(* CODESYS project elevator_project.project

Project tree, tasks and I/O mapping:
  Device : CODESYS Control Win V3, 3S - Smart Software Solutions GmbH, order no. 305021, version 3.5.9.40
    application Application
      libraries: Standard, * (System)
      task MainTask (cyclic, interval t#20ms, priority 1) calls PLC_PRG
      task VISU_TASK (cyclic, interval 100 ms, priority 31) calls VisuElems.Visu_Prg
      program PLC_PRG [SFC]: Init_entry, Init_active, GoTo_active, Idle_entry, Idle_exit, UpdateDesireFloor_active, UP_entry, DOWN_entry, UP_active, DOWN_active, Idle_active, Listener
      global variables GVL
      visualisation Visualization
  libraries: VisuSymbols, 3.5.8.0 (System)
  text list GlobalTextList
*)

// Device/Application/GVL
{attribute 'qualified_only'}
VAR_GLOBAL
	AtLevel1: BOOL;
	AtLevel2: BOOL;
	AtLevel3: BOOL;
	
	overweight: BOOL;
	
	Bottom: BOOL;
	Top: BOOL;
	
	Call1: BOOL;
	Call2: BOOL;
	Call3: BOOL;
	
	GoLevel1: BOOL;
	GoLevel2: BOOL;
	GoLevel3: BOOL;
	
	goDown: BOOL;
	goUp: BOOL;
	
	// Code
	calls: ARRAY[1..3] OF BOOL;
	i: INT;
	
	NOKButton: BOOL;
	goingUp: BOOL;
	goingDown: BOOL;
	desiredFloor: INT:=1;
	currentFloor: INT:=2;
	MAXFLOOR: INT:=3;
	
	useless: BOOL;
	
	openDahDoor: BOOL;
	arrived: BOOL;
	
	Done: BOOL;
	
	// State
	InitOk: BOOL;
	busy: BOOL;
	emergency: BOOL;
	request: BOOL;
END_VAR

// Device/Application/PLC_PRG
PROGRAM PLC_PRG
VAR
END_VAR
VAR // added by the converter: edge detectors and wires of the graphical bodies
    _w1, _w3, _w5, _w6, _w8, _w9, _w10, _w11 : BOOL;
    _w2, _w4, _w7 : INT;
END_VAR

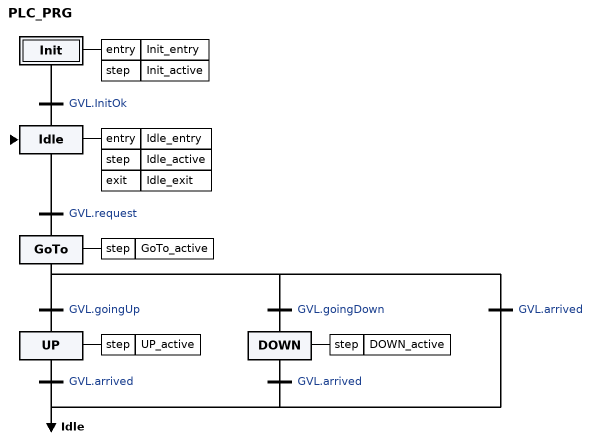
INITIAL_STEP Init:
    Init_entry(P1);  // entry action
    Init_active(N);  // step action
END_STEP
TRANSITION FROM Init TO Idle
    := GVL.InitOk;
END_TRANSITION
STEP Idle:
    Idle_entry(P1);  // entry action
    Idle_active(N);  // step action
    Idle_exit(P0);  // exit action
END_STEP
TRANSITION FROM Idle TO GoTo
    := GVL.request;
END_TRANSITION
STEP GoTo:
    GoTo_active(N);  // step action
END_STEP
TRANSITION FROM GoTo TO UP
    := GVL.goingUp;
END_TRANSITION
STEP UP:
    UP_active(N);  // step action
END_STEP
TRANSITION FROM UP TO Idle
    := GVL.arrived;
END_TRANSITION
TRANSITION FROM GoTo TO DOWN
    := GVL.goingDown;
END_TRANSITION
STEP DOWN:
    DOWN_active(N);  // step action
END_STEP
TRANSITION FROM DOWN TO Idle
    := GVL.arrived;
END_TRANSITION
TRANSITION FROM GoTo TO Idle
    := GVL.arrived;
END_TRANSITION

ACTION Init_entry:
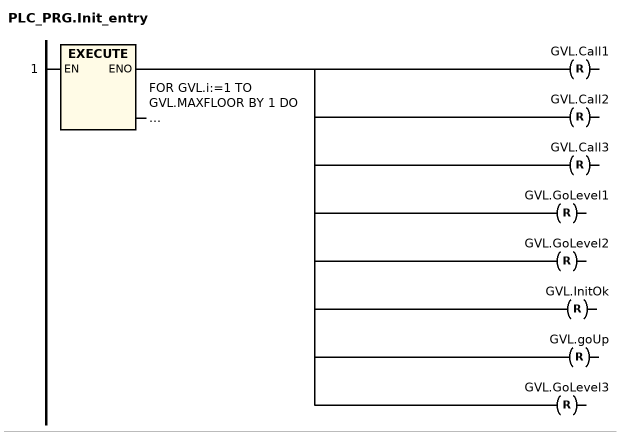
// NETWORK 1
FOR GVL.i:=1 TO GVL.MAXFLOOR BY 1 DO
	GVL.calls[GVL.i]:=FALSE;
END_FOR;
GVL.Call1 R= TRUE;
GVL.Call2 R= TRUE;
GVL.Call3 R= TRUE;
GVL.GoLevel1 R= TRUE;
GVL.GoLevel2 R= TRUE;
GVL.InitOk R= TRUE;
GVL.goUp R= TRUE;
GVL.GoLevel3 R= TRUE;
END_ACTION

ACTION Init_active:
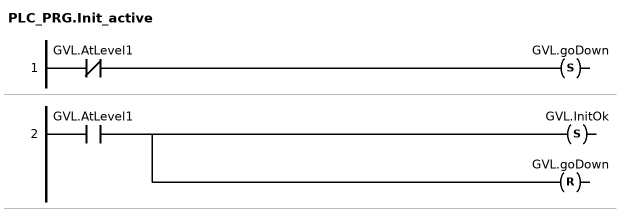
// NETWORK 1
GVL.goDown S= NOT GVL.AtLevel1;

// NETWORK 2
_w1 := GVL.AtLevel1;
GVL.InitOk S= _w1;
GVL.goDown R= _w1;
END_ACTION

ACTION GoTo_active:
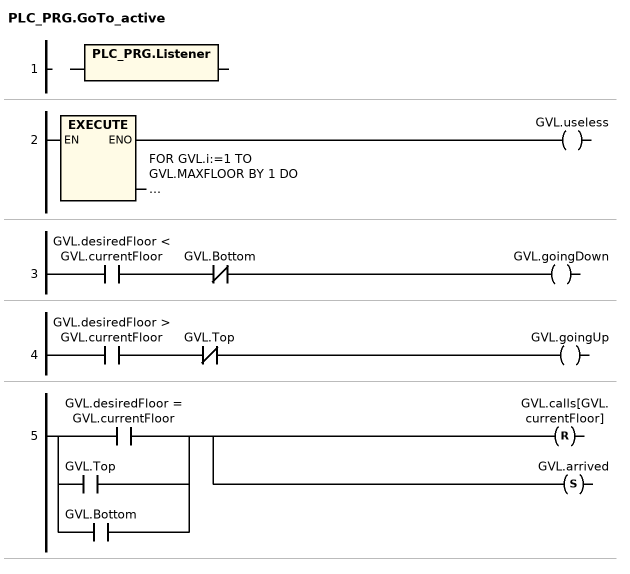
// NETWORK 1
PLC_PRG.Listener();

// NETWORK 2
FOR GVL.i:=1 TO GVL.MAXFLOOR BY 1 DO
	IF (GVL.calls[GVL.i]=TRUE) THEN
		GVL.desiredFloor:=GVL.i;
	END_IF
END_FOR;
GVL.useless := TRUE;

// NETWORK 3
GVL.goingDown := (GVL.desiredFloor < GVL.currentFloor) AND NOT GVL.Bottom;

// NETWORK 4
GVL.goingUp := (GVL.desiredFloor > GVL.currentFloor) AND NOT GVL.Top;

// NETWORK 5
_w2 := (GVL.desiredFloor = GVL.currentFloor) OR GVL.Top OR GVL.Bottom;
GVL.calls[GVL.currentFloor] R= _w2;
GVL.arrived S= _w2;
END_ACTION

ACTION Idle_entry:
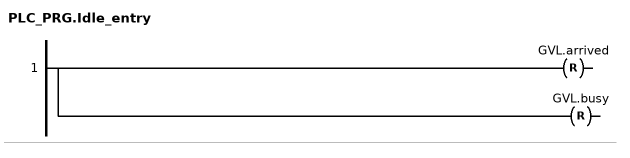
// NETWORK 1
GVL.arrived R= TRUE;
GVL.busy R= TRUE;
END_ACTION

ACTION Idle_exit:
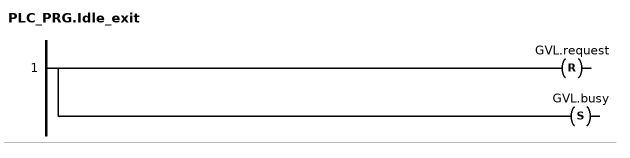
// NETWORK 1
GVL.request R= TRUE;
GVL.busy S= TRUE;
END_ACTION

ACTION UpdateDesireFloor_active:
// NETWORK 1
END_ACTION

ACTION UP_entry:
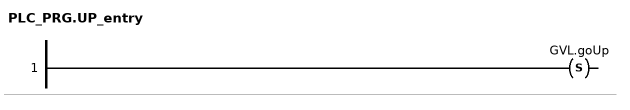
// NETWORK 1
GVL.goUp S= TRUE;
END_ACTION

ACTION DOWN_entry:
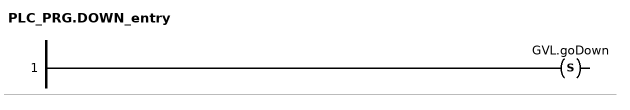
// NETWORK 1
GVL.goDown S= TRUE;
END_ACTION

ACTION UP_active:
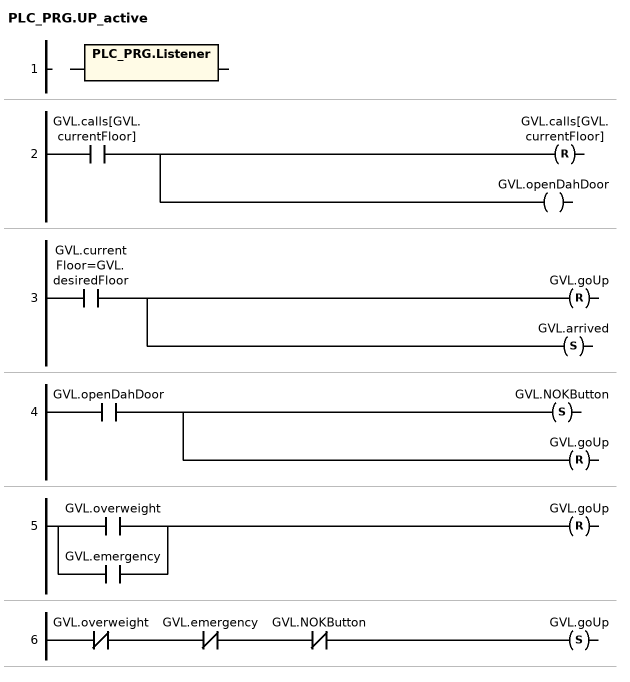
// NETWORK 1
PLC_PRG.Listener();

// NETWORK 2
_w3 := GVL.calls[GVL.currentFloor];
GVL.calls[GVL.currentFloor] R= _w3;
GVL.openDahDoor := _w3;

// NETWORK 3
_w4 := GVL.currentFloor=GVL.desiredFloor;
GVL.goUp R= _w4;
GVL.arrived S= _w4;

// NETWORK 4
_w5 := GVL.openDahDoor;
GVL.NOKButton S= _w5;
GVL.goUp R= _w5;

// NETWORK 5
GVL.goUp R= GVL.overweight OR GVL.emergency;

// NETWORK 6
GVL.goUp S= NOT GVL.overweight AND NOT GVL.emergency AND NOT GVL.NOKButton;
END_ACTION

ACTION DOWN_active:
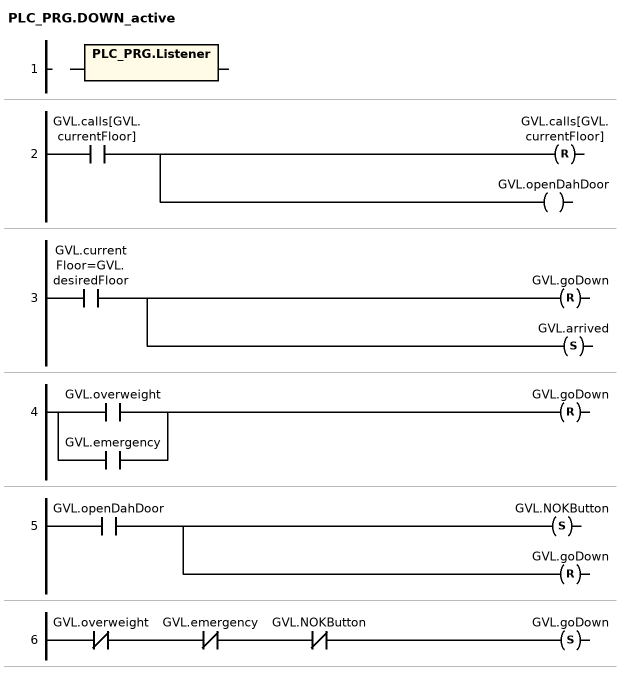
// NETWORK 1
PLC_PRG.Listener();

// NETWORK 2
_w6 := GVL.calls[GVL.currentFloor];
GVL.calls[GVL.currentFloor] R= _w6;
GVL.openDahDoor := _w6;

// NETWORK 3
_w7 := GVL.currentFloor=GVL.desiredFloor;
GVL.goDown R= _w7;
GVL.arrived S= _w7;

// NETWORK 4
GVL.goDown R= GVL.overweight OR GVL.emergency;

// NETWORK 5
_w8 := GVL.openDahDoor;
GVL.NOKButton S= _w8;
GVL.goDown R= _w8;

// NETWORK 6
GVL.goDown S= NOT GVL.overweight AND NOT GVL.emergency AND NOT GVL.NOKButton;
END_ACTION

ACTION Idle_active:
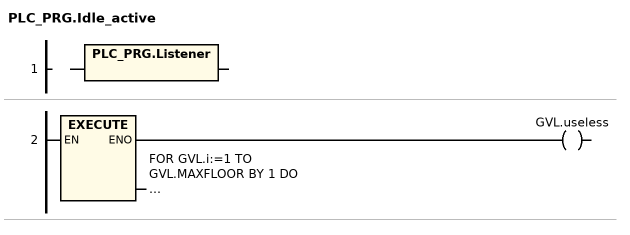
// NETWORK 1
PLC_PRG.Listener();

// NETWORK 2
FOR GVL.i:=1 TO GVL.MAXFLOOR BY 1 DO
	IF (GVL.calls[GVL.i]=TRUE) THEN
		GVL.request:=TRUE;
	END_IF
END_FOR;
GVL.useless := TRUE;
END_ACTION

ACTION Listener:
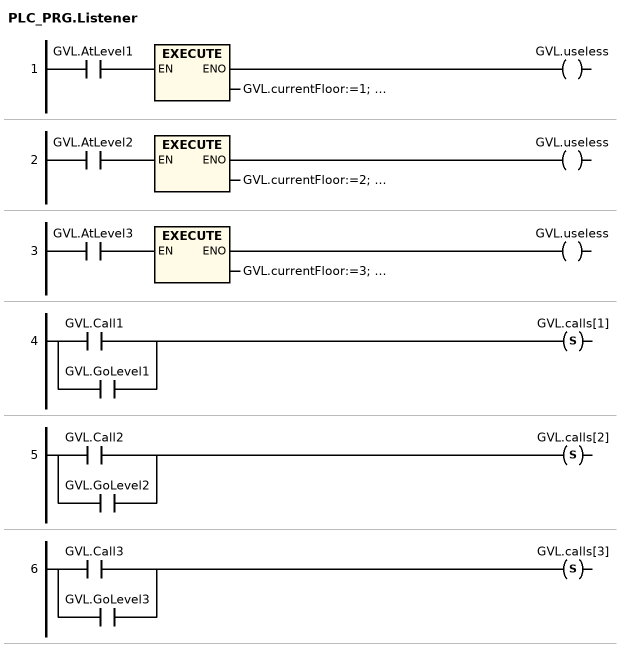
// NETWORK 1
_w9 := GVL.AtLevel1;
IF _w9 THEN GVL.currentFloor:=1; END_IF
GVL.useless := _w9;

// NETWORK 2
_w10 := GVL.AtLevel2;
IF _w10 THEN GVL.currentFloor:=2; END_IF
GVL.useless := _w10;

// NETWORK 3
_w11 := GVL.AtLevel3;
IF _w11 THEN GVL.currentFloor:=3; END_IF
GVL.useless := _w11;

// NETWORK 4
GVL.calls[1] S= GVL.Call1 OR GVL.GoLevel1;

// NETWORK 5
GVL.calls[2] S= GVL.Call2 OR GVL.GoLevel2;

// NETWORK 6
GVL.calls[3] S= GVL.Call3 OR GVL.GoLevel3;
END_ACTION

END_PROGRAM

// Device/Application/Visualization
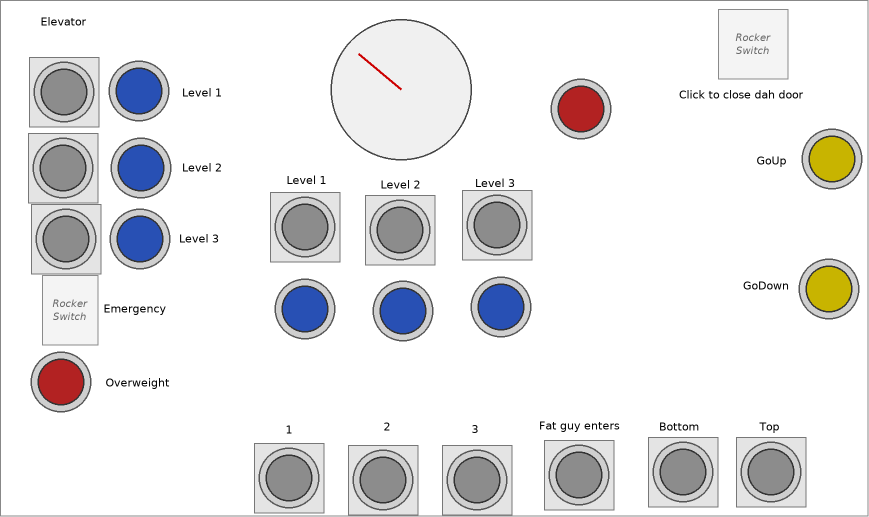
VISUALIZATION Visualization  // 869x517
    Label (30,7 67x30), "Elevator"
    Label (271,164 71x33), "Level 1"
    Label (347,172 107x26), "Level 2"
    Label (438,171 114x25), "Level 3"
    PushSwitch (29,57 70x70), variable: GVL.GoLevel1, behaviour: TAP, style: Switch-PushSwitch-Gray
    PushSwitch (28,133 70x70), variable: GVL.GoLevel2, behaviour: TAP, style: Switch-PushSwitch-Gray
    PushSwitch (462,190 70x70), variable: GVL.Call3, behaviour: TAP, style: Switch-PushSwitch-Gray
    PushSwitch (365,195 70x70), variable: GVL.Call2, behaviour: TAP, style: Switch-PushSwitch-Gray
    PushSwitch (270,192 70x70), variable: GVL.Call1, behaviour: TAP, style: Switch-PushSwitch-Gray
    PushSwitch (31,204 70x70), variable: GVL.GoLevel3, behaviour: TAP, style: Switch-PushSwitch-Gray
    Lamp1 (466,272 70x70), variable: GVL.calls[3], style: Lamp-Lamp1-Blue
    Lamp1 (368,276 70x70), variable: GVL.calls[2], style: Lamp-Lamp1-Blue
    Lamp1 (270,274 70x70), variable: GVL.calls[1], style: Lamp-Lamp1-Blue
    Lamp1 (105,204 70x70), variable: GVL.calls[3], style: Lamp-Lamp1-Blue
    Lamp1 (106,133 70x70), variable: GVL.calls[2], style: Lamp-Lamp1-Blue
    Lamp1 (104,56 70x70), variable: GVL.calls[1], style: Lamp-Lamp1-Blue
    Lamp1 (26,347 70x70), variable: GVL.overweight, style: Lamp-Lamp1-Red
    Lamp1 (546,74 70x70), variable: GVL.busy, style: Lamp-Lamp1-Red
    Label (94,368 87x30), "Overweight"
    Label (95,294 80x30), "Emergency"
    Label (162,78 80x30), "Level 1"
    Label (162,153 80x30), "Level 2"
    Label (159,224 80x30), "Level 3"
    Meter180 (276,19 250x141), value: GVL.currentFloor, style: Meter-Meter180-Gray, scale format: %.1f, scale 1..3
    PushSwitch (254,443 70x70), variable: GVL.AtLevel1, behaviour: TOGGLE, style: Switch-PushSwitch-Gray
    PushSwitch (348,445 70x70), variable: GVL.AtLevel2, behaviour: TOGGLE, style: Switch-PushSwitch-Gray
    PushSwitch (442,445 70x70), variable: GVL.AtLevel3, behaviour: TOGGLE, style: Switch-PushSwitch-Gray
    Lamp1 (797,124 70x70), variable: GVL.goUp, style: Lamp-Lamp1-Yellow
    Lamp1 (794,254 70x70), variable: GVL.goDown, style: Lamp-Lamp1-Yellow
    Label (738,146 67x30), "GoUp"
    Label (732,271 68x30), "GoDown"
    RockerSwitch (42,275 56x70), variable: GVL.emergency, behaviour: TOGGLE, style: Switch-RockerSwitch-Gray
    PushSwitch (544,440 70x70), variable: GVL.overweight, behaviour: TOGGLE, style: Switch-PushSwitch-Gray
    Label (532,411 95x30), "Fat guy enters"
    Label (271,415 36x30), "1"
    Label (368,412 38x30), "2"
    Label (448,415 54x29), "3"
    PushSwitch (736,437 70x70), variable: GVL.Top, behaviour: TOGGLE, style: Switch-PushSwitch-Gray
    PushSwitch (648,437 70x70), variable: GVL.Bottom, behaviour: TOGGLE, style: Switch-PushSwitch-Gray
    Label (650,412 58x30), "Bottom"
    Label (744,412 51x30), "Top"
    RockerSwitch (718,9 70x70), variable: GVL.NOKButton, behaviour: TOGGLE, style: Switch-RockerSwitch-Gray
    Label (666,80 150x30), "Click to close dah door"
END_VISUALIZATION
